// SIMATIC S7-200 project (STEP 7-Micro/WIN), CPU 224 REL 02.01

SYMBOL_TABLE Command
hhhmi_to_plc     VW401
aaa_to_plc       VW402
dor_baraye_1_doff VW320
second_PLC       VW318
minute_PLC       VW316
hour_PLC         VW314
RPM_mani_Cylinder_HMI VW312    // analog_output
RPM_Doffer_Int   VW310    // rpm
RPM_main_Int     VW308    // rpm
RPM_Feed_in_HMI  VW306    // analog_output
RPM_Coiler_In_HMI VW304    // analog_output
RPM_Sec_Cyli_in_HMI VW302    // analog_output
RPM_Doffer_in_HMI VW300    // analog_output
Minute_shiftC    VW248    // amar
hour_shiftC      VW246    // amar
minute_shiftB    VW244    // amar
Lengh            VW242    // doff
max_rpm_SecCylindr VW240    // analog_output
max_rpm_feeder   VW238    // analog_output
max_rpm_coiler   VW236    // analog_output
max_rpm_doffer_cylinder VW234    // analog_output
max_rpm_main_cylinder VW232    // rpm
zaribe_asli_doffer VW230    // rpm
hour_shiftB      VW228    // amar
doff_in_shiftc   VW224    // amar
Minute_ShiftA    VW222    // amar
doff_in_shiftB   VW218    // amar
hour_ShiftA      VW216    // amar
doff_in_shiftA   VW212    // amar
enter_rpm_in_HMI VW210    // analog_output
Zaribe_Asli      VW208    // rpm
Zaribe_Fed       VW206    // analog_output
Zaribe_Coi       VW204    // analog_output
Zaribe_Sec       VW202    // analog_output
Zaribe_Doff      VW200    // analog_output
zaribe_asli2     VD800
leng_for_1rotate_coiler VD720    // doff
Vazne_kole_C     VD712
Vazne_kole_B     VD708
vazne_kole_A     VD704
nomre_fetile     VD700
RPM_Main         VD504
RPM_Doffer       VD500
reset_metal      V104.1
metal_blink_hmi  V104.0
metal_hmi        V103.7
fault            V103.6
coiler_fault     V103.5   // startstop
Metal            V103.4   // startstop
Pulse            V103.3   // pulse_700ms
Doff_Lamp_F      V103.2   // doff
reset_lengh      V103.1   // doff
reset_Amar       V103.0
photocell_coiler_fault V101.6
key_stop_pushed  V101.1   // alarm
Machin_Fault     V101.0   // alarm
OL_Za_F          V100.7   // alarm
OL_ap_F          V100.6   // alarm
OL_Chane_F       V100.5   // alarm
Fauklt_CoilerDrive_F V100.4   // alarm
Fault_FeederDrive_F V100.3   // alarm
Fault_DofferDrive_F V100.2   // alarm
Fault_secDrive_F V100.1   // alarm
fault_mainDrive_F V100.0   // alarm
delay_300ms      T63
metal            T62
timer_for_metal  T61
time_for_push_stop T60
timer_for_coilerfult T59      // start_stop
timer_for_metaldetector T58      // start_stop
Timer57          T57
Timer56          T56
delay            T55      // doff
timer_for_reset_lengh T54      // doff
Timer_for_fan2   T53      // fan
timer_for_fan1   T52      // fan
Stop_Apron       T51      // hopper
for_start_apron  T50      // hopper
Ajir_metal       Q2.5
Fan2             Q2.4
Orange_Lamp      Q2.2
Red_Lamp         Q2.1
Green_Lamp       Q2.0
Feeder_Reverse   Q1.1
Fan1             Q1.0
Zanandeh         Q0.7
Apron            Q0.6
motor_Change_Doff Q0.5
motor_Feeder_Forward Q0.4
motor_Coiler     Q0.3
motor_Doffer     Q0.2
Secondary        Q0.1
Main_Sylinder    Q0.0
Chaper_fault     I2.5
manual_doff      I2.4
OL_Zanandeh      I2.3
OL_Apron         I2.2
OL_change_doff   I2.1
Photocell        I2.0
photocell_coiler I1.5
Fault_Feeder_Drive I1.4
Fault_Coiler_Drive I1.3
Fault_Doffer_Drive I1.2
Fault_Secondary_Drive I1.1
Fault_MainDrive  I1.0
MetalDetector    I0.7
Motor_Doff_SW    I0.5
Emergency        I0.4
Stopp            I0.3
Start            I0.2
Product_SW       I0.1
Hour_counter     C4       // amar
Minute_Counter   C3       // amar
Scond_counter    C2
doff_counter     C1       // amar
lengh_counter    C0
An_Feeder        AQW8
An_Doffer        AQW6
An_Coiler        AQW4
An_Seco_Syl      AQW2
An_Main_Syl      AQW0
                 ?0_40_0  // pulse_700ms
                 ?0_40_0  // pulse_700ms
                 ?0_40_0  // amar
                 ?0_40_0  // amar
                 ?0_40_0  // amar
END_SYMBOL_TABLE

ORGANIZATION_BLOCK Main:OB1
TITLE=vw200 & vw300  -------   vd700 & vd900 ======>> retentive
// vw300 & vw & vw500   ,   vd500 & vd700 =====>not retentive
// vw100 & vw200  ====>> flag
BEGIN
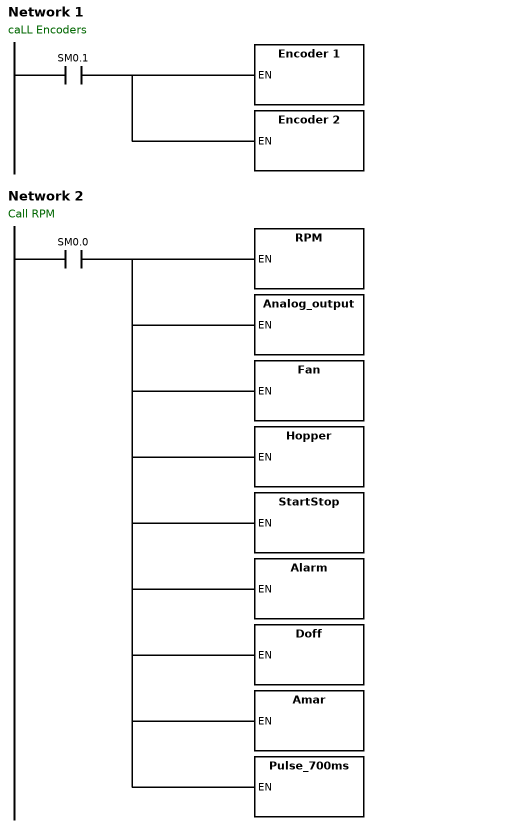
Network 1
// caLL Encoders
LD     SM0.1
CALL   Encoder 1:SBR1
CALL   Encoder 2:SBR2
Network 2
// Call RPM
LD     SM0.0
CALL   RPM:SBR3
CALL   Analog_output:SBR4
CALL   Fan:SBR5
CALL   Hopper:SBR6
CALL   StartStop:SBR8
CALL   Alarm:SBR7
CALL   Doff:SBR9
CALL   Amar:SBR10
CALL   Pulse_700ms:SBR11
END_ORGANIZATION_BLOCK

SUBROUTINE_BLOCK PtoRPM:SBR0
TITLE=子程序注释
VAR_INPUT
Plus:DWORD;	// LD0 
Lines:DWORD;	// LD4 
END_VAR
VAR_IN_OUT
Plusbefore:DWORD;	// LD8 
END_VAR
VAR_OUTPUT
RpmofEncoder:DWORD;	// LD12 
END_VAR
BEGIN
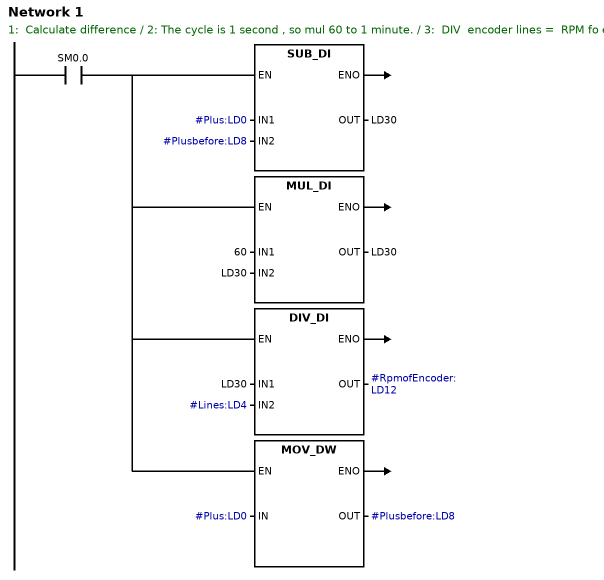
Network 1
// 1:  Calculate difference
// 2: The cycle is 1 second , so mul 60 to 1 minute.
// 3:  DIV  encoder lines =  RPM fo encoder
// 4: save plus to plusbefore
LD     SM0.0
MOVD   #Plus:LD0, LD30
-D     #Plusbefore:LD8, LD30
*D     60, LD30
MOVD   LD30, #RpmofEncoder:LD12
/D     #Lines:LD4, #RpmofEncoder:LD12
MOVD   #Plus:LD0, #Plusbefore:LD8
END_SUBROUTINE_BLOCK

SUBROUTINE_BLOCK Encoder 1:SBR1
TITLE=
BEGIN
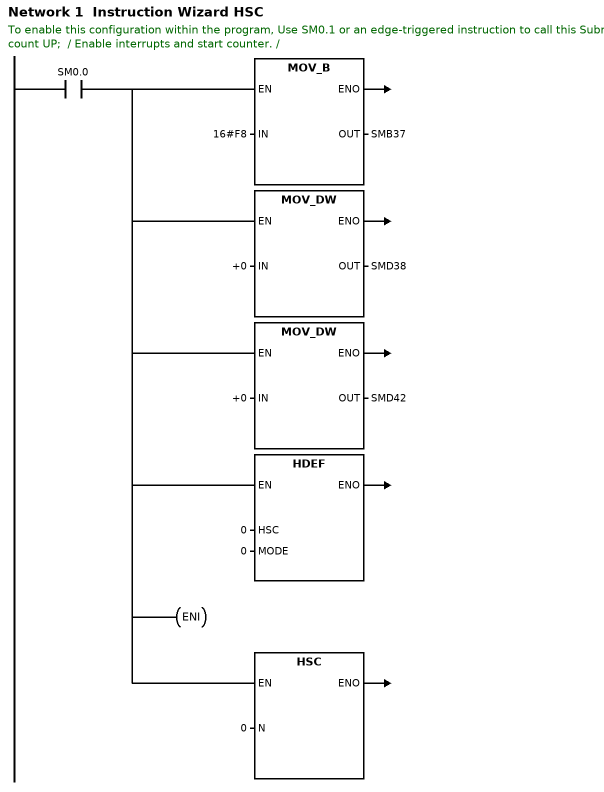
Network 1 // Instruction Wizard HSC
// To enable this configuration within the program, Use SM0.1 or an edge-triggered instruction to call this Subroutine once from the MAIN program block.  
// Configure HC0 for Mode 0; CV = 0; PV = 0; count UP; 
// Enable interrupts and start counter.
// 
//Set control bits: count UP; enabled; 
//Load CV
//Load PV
LD     SM0.0
MOVB   16#F8, SMB37
MOVD   +0, SMD38
MOVD   +0, SMD42
HDEF   0, 0
ENI
HSC    0
END_SUBROUTINE_BLOCK

SUBROUTINE_BLOCK Encoder 2:SBR2
TITLE=
BEGIN
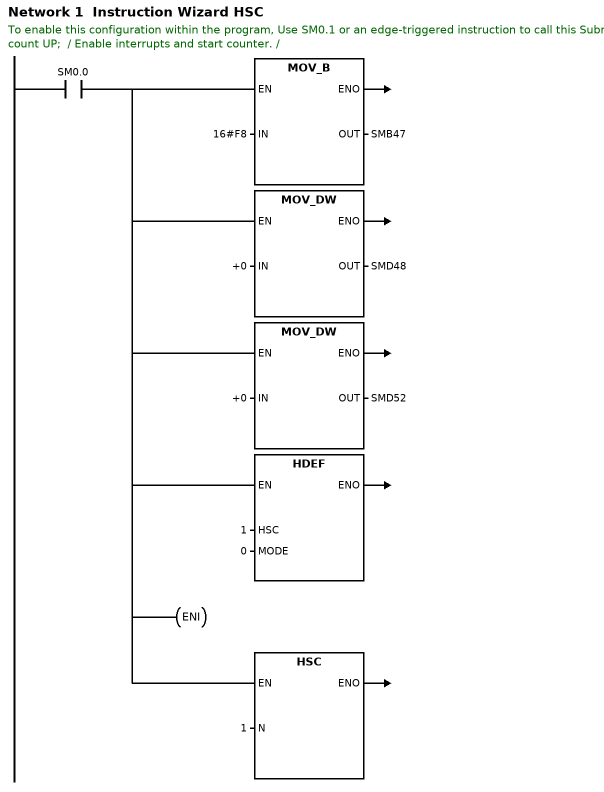
Network 1 // Instruction Wizard HSC
// To enable this configuration within the program, Use SM0.1 or an edge-triggered instruction to call this Subroutine once from the MAIN program block.  
// Configure HC1 for Mode 0; CV = 0; PV = 0; count UP; 
// Enable interrupts and start counter.
// 
//Set control bits: count UP; enabled; 
//Load CV
//Load PV
LD     SM0.0
MOVB   16#F8, SMB47
MOVD   +0, SMD48
MOVD   +0, SMD52
HDEF   1, 0
ENI
HSC    1
END_SUBROUTINE_BLOCK

SUBROUTINE_BLOCK RPM:SBR3
TITLE=SUBROUTINE COMMENTS
VAR
rpm1:REAL;	// LD0 
rpm2:REAL;	// LD4 
rpm11:REAL;	// LD8 
rpm21:REAL;	// LD12 
END_VAR
BEGIN
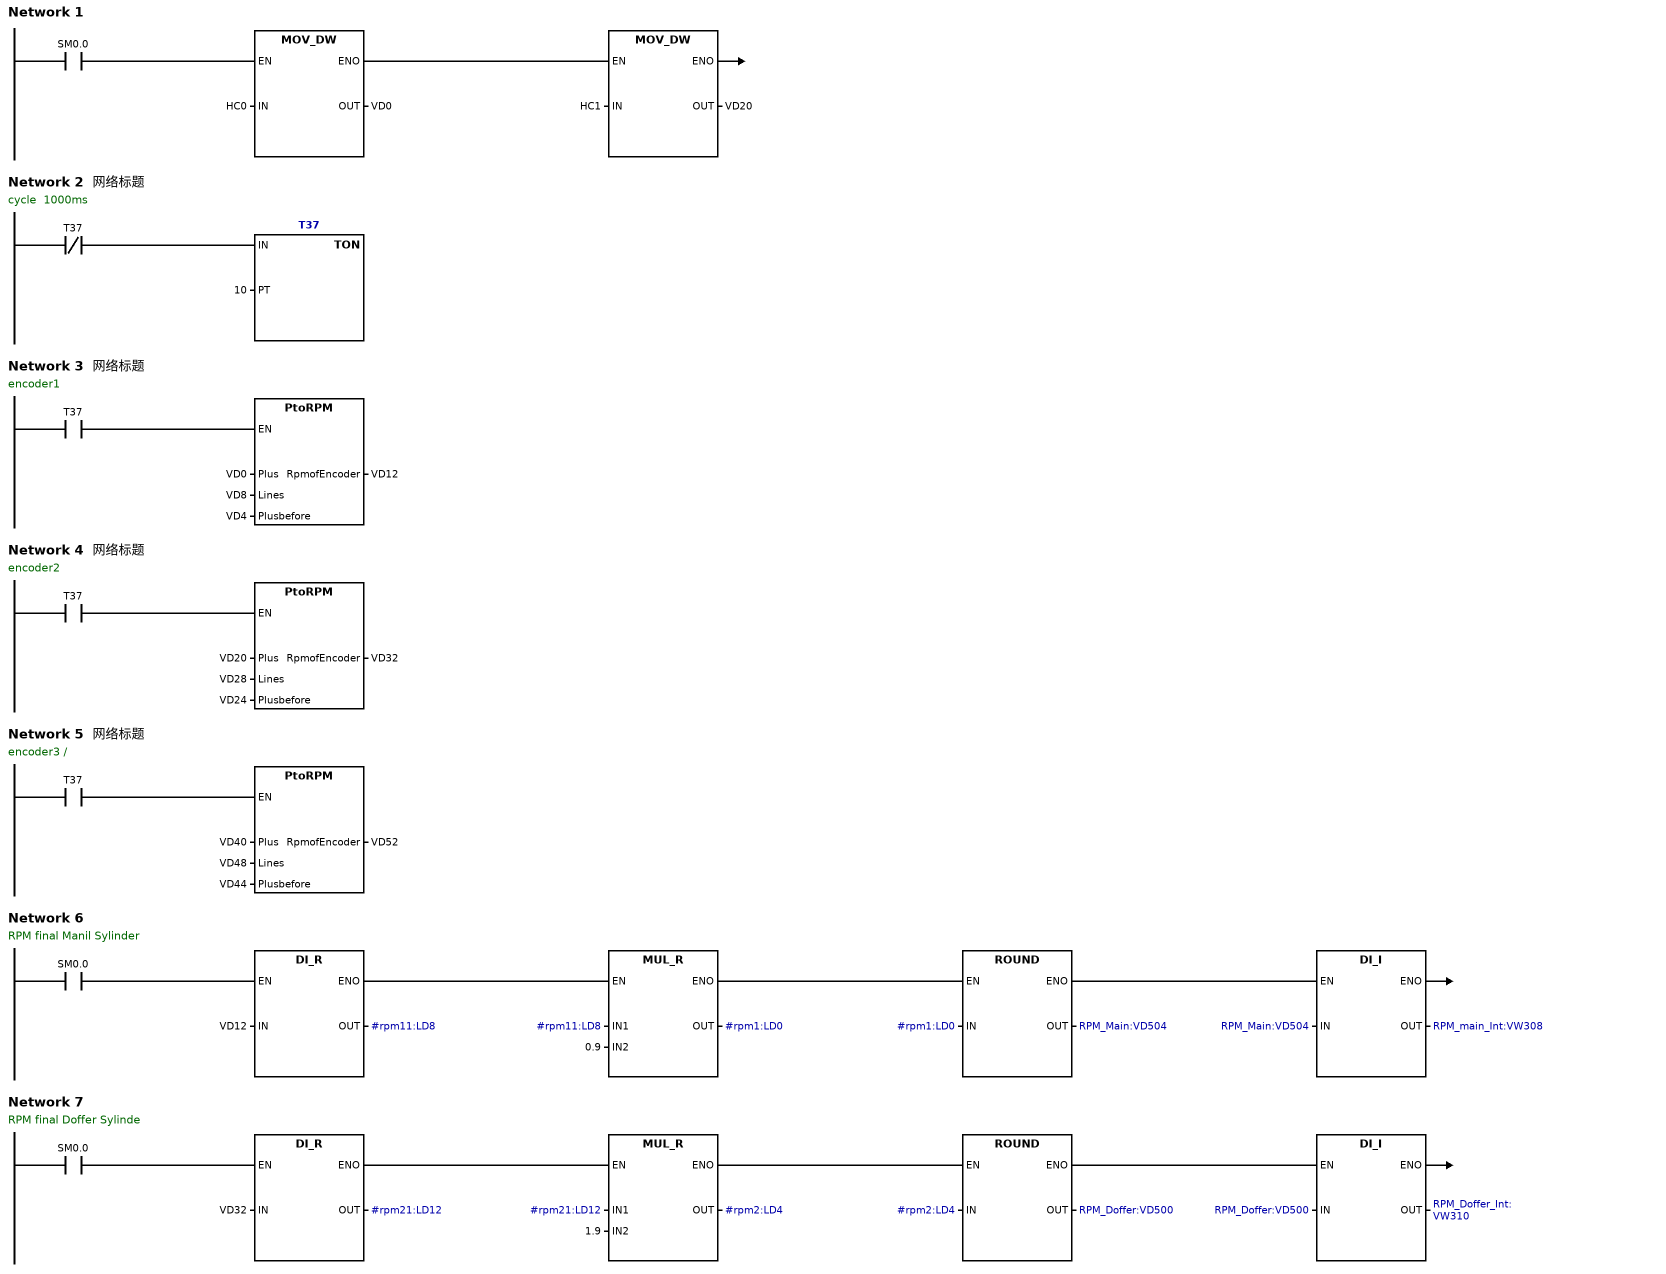
Network 1
LD     SM0.0
MOVD   HC0, VD0
AENO
MOVD   HC1, VD20
Network 2 // 网络标题
// cycle  1000ms 
LDN    T37
TON    T37, 10
Network 3 // 网络标题
// encoder1
LD     T37
CALL   PtoRPM:SBR0, VD0, VD8, VD4, VD12
Network 4 // 网络标题
// encoder2
LD     T37
CALL   PtoRPM:SBR0, VD20, VD28, VD24, VD32
Network 5 // 网络标题
// encoder3
// 
LD     T37
CALL   PtoRPM:SBR0, VD40, VD48, VD44, VD52
Network 6
// RPM final Manil Sylinder
LD     SM0.0
DTR    VD12, #rpm11:LD8
AENO
MOVR   #rpm11:LD8, #rpm1:LD0
AENO
*R     0.9, #rpm1:LD0
AENO
ROUND  #rpm1:LD0, RPM_Main:VD504
AENO
DTI    RPM_Main:VD504, RPM_main_Int:VW308
Network 7
// RPM final Doffer Sylinde
LD     SM0.0
DTR    VD32, #rpm21:LD12
AENO
MOVR   #rpm21:LD12, #rpm2:LD4
AENO
*R     1.9, #rpm2:LD4
AENO
ROUND  #rpm2:LD4, RPM_Doffer:VD500
AENO
DTI    RPM_Doffer:VD500, RPM_Doffer_Int:VW310
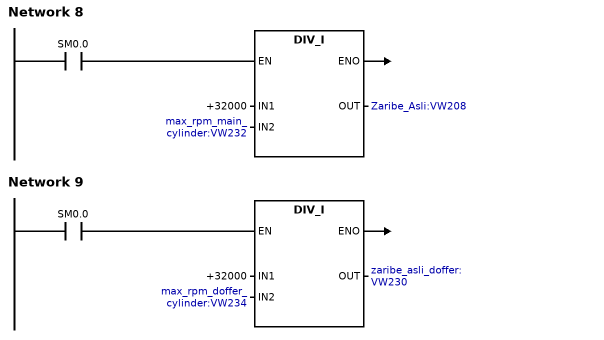
Network 8
LD     SM0.0
MOVW   +32000, Zaribe_Asli:VW208
/I     max_rpm_main_cylinder:VW232, Zaribe_Asli:VW208
Network 9
LD     SM0.0
MOVW   +32000, zaribe_asli_doffer:VW230
/I     max_rpm_doffer_cylinder:VW234, zaribe_asli_doffer:VW230
END_SUBROUTINE_BLOCK

SUBROUTINE_BLOCK Analog_output:SBR4
TITLE=SUBROUTINE COMMENTS
VAR
rpm_doff1:DINT;	// LD0 
rpm_doff2:DINT;	// LD4 
rpm_doff3:INT;	// LW8 
rpm_sec1:INT;	// LW10 
rpm_sec2:INT;	// LW12 
rpm_sec3:INT;	// LW14 
rpm_coil1:INT;	// LW16 
rpm_coil2:INT;	// LW18 
rpm_coil3:INT;	// LW20 
ADD:INT;	// LW22 
rpm_feed2:INT;	// LW24 
rpm_feed3:INT;	// LW26 
speed_main:INT;	// LW28 
main_hmi1:INT;	// LW30 
main_hmi2:INT;	// LW32 
dofer_hmi1:INT;	// LW34 
dofer_hmi2:INT;	// LW36 
sec_hmi1:INT;	// LW38 
sec_hmi2:INT;	// LW40 
coiler_hmi1:INT;	// LW42 
coiler_hmi2:INT;	// LW44 
feeder_hmi1:INT;	// LW46 
feeder_hmi2:INT;	// LW48 
rmp_doffer1:DINT;	// LD50 
rpm_doffer2:DINT;	// LD54 
END_VAR
BEGIN
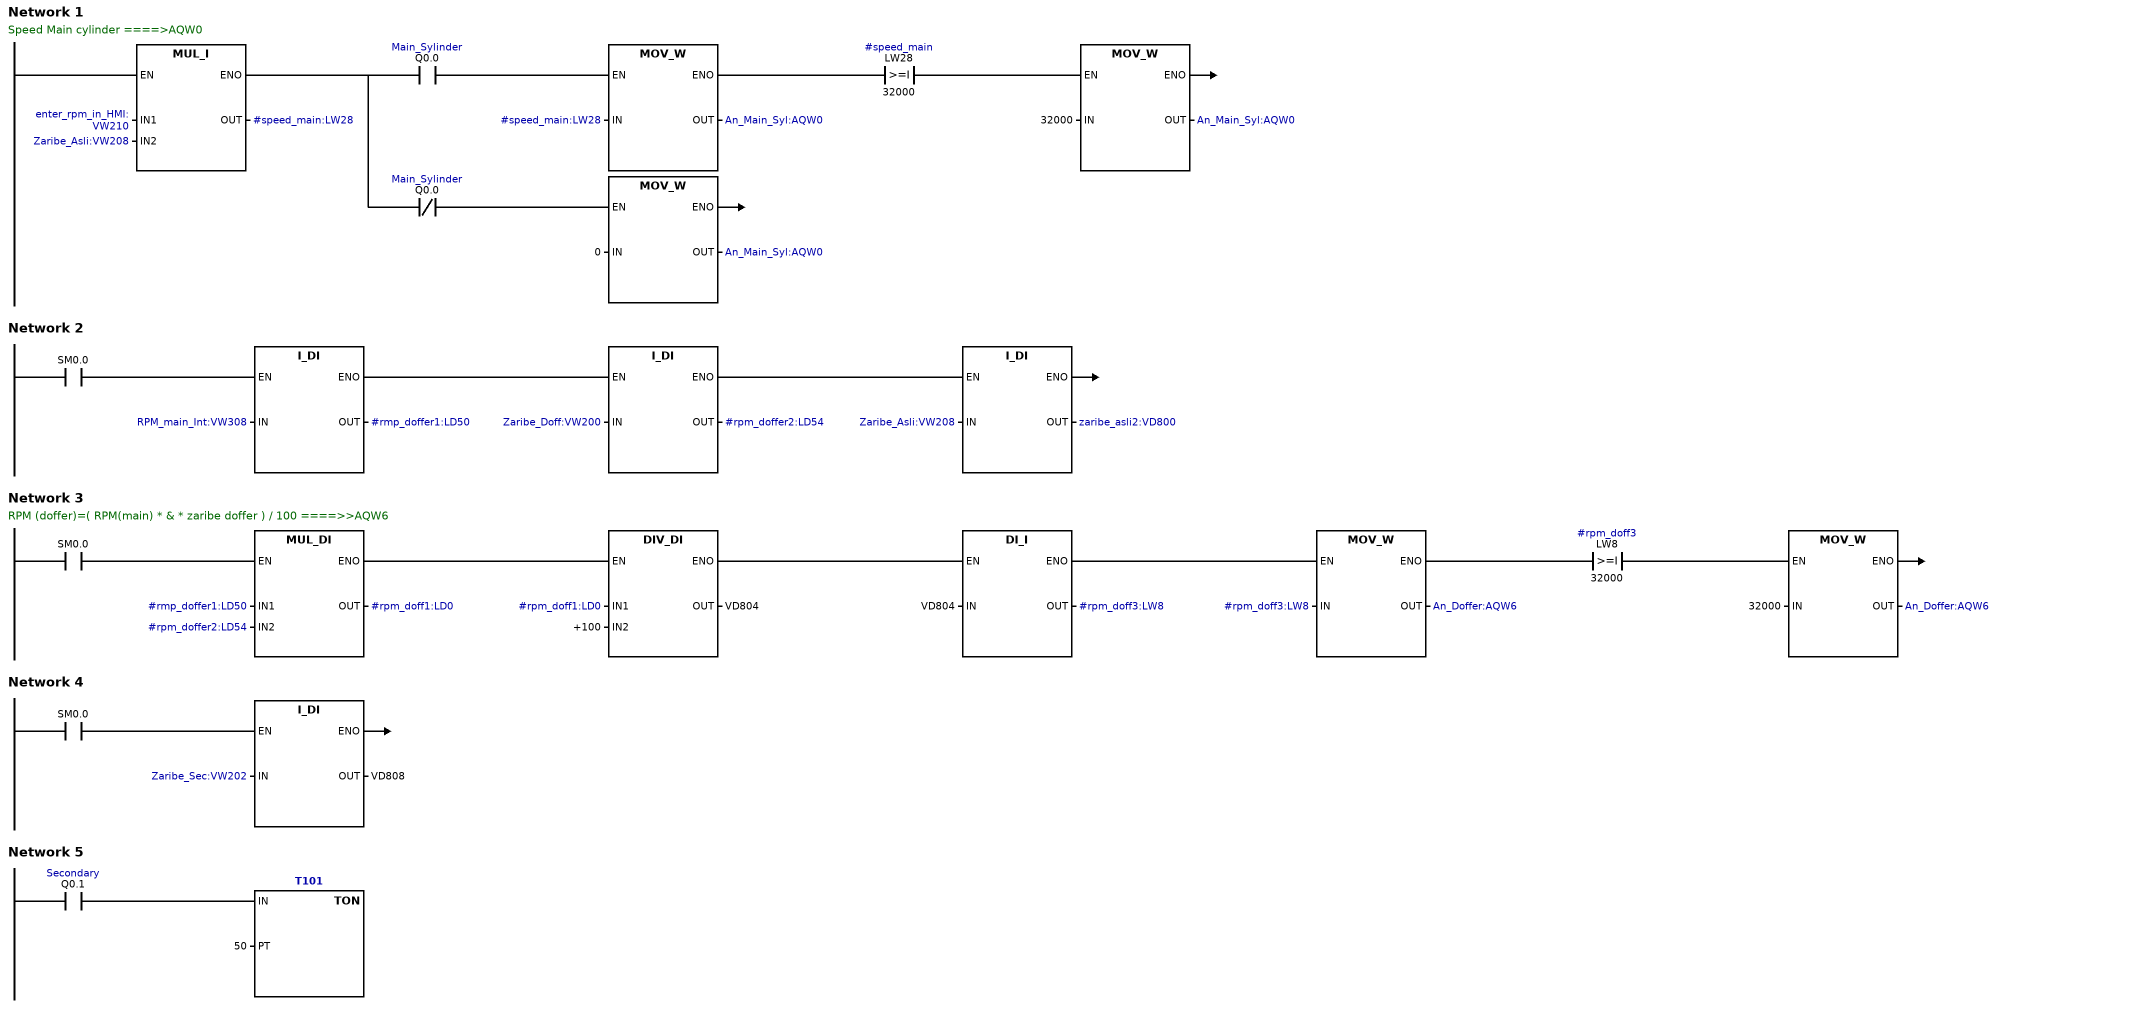
Network 1
// Speed Main cylinder ====>AQW0
MOVW   enter_rpm_in_HMI:VW210, #speed_main:LW28
AENO
*I     Zaribe_Asli:VW208, #speed_main:LW28
AENO
LPS
A      Main_Sylinder:Q0.0
MOVW   #speed_main:LW28, An_Main_Syl:AQW0
AENO
AW>=   #speed_main:LW28, 32000
MOVW   32000, An_Main_Syl:AQW0
LPP
AN     Main_Sylinder:Q0.0
MOVW   0, An_Main_Syl:AQW0
Network 2
LD     SM0.0
ITD    RPM_main_Int:VW308, #rmp_doffer1:LD50
AENO
ITD    Zaribe_Doff:VW200, #rpm_doffer2:LD54
AENO
ITD    Zaribe_Asli:VW208, zaribe_asli2:VD800
Network 3
// RPM (doffer)=( RPM(main) * & * zaribe doffer ) / 100 ====>>AQW6
LD     SM0.0
MOVD   #rmp_doffer1:LD50, #rpm_doff1:LD0
AENO
*D     #rpm_doffer2:LD54, #rpm_doff1:LD0
AENO
MOVD   #rpm_doff1:LD0, VD804
AENO
/D     +100, VD804
AENO
DTI    VD804, #rpm_doff3:LW8
AENO
MOVW   #rpm_doff3:LW8, An_Doffer:AQW6
AENO
AW>=   #rpm_doff3:LW8, 32000
MOVW   32000, An_Doffer:AQW6
Network 4
LD     SM0.0
ITD    Zaribe_Sec:VW202, VD808
Network 5
LD     Secondary:Q0.1
TON    T101, 50
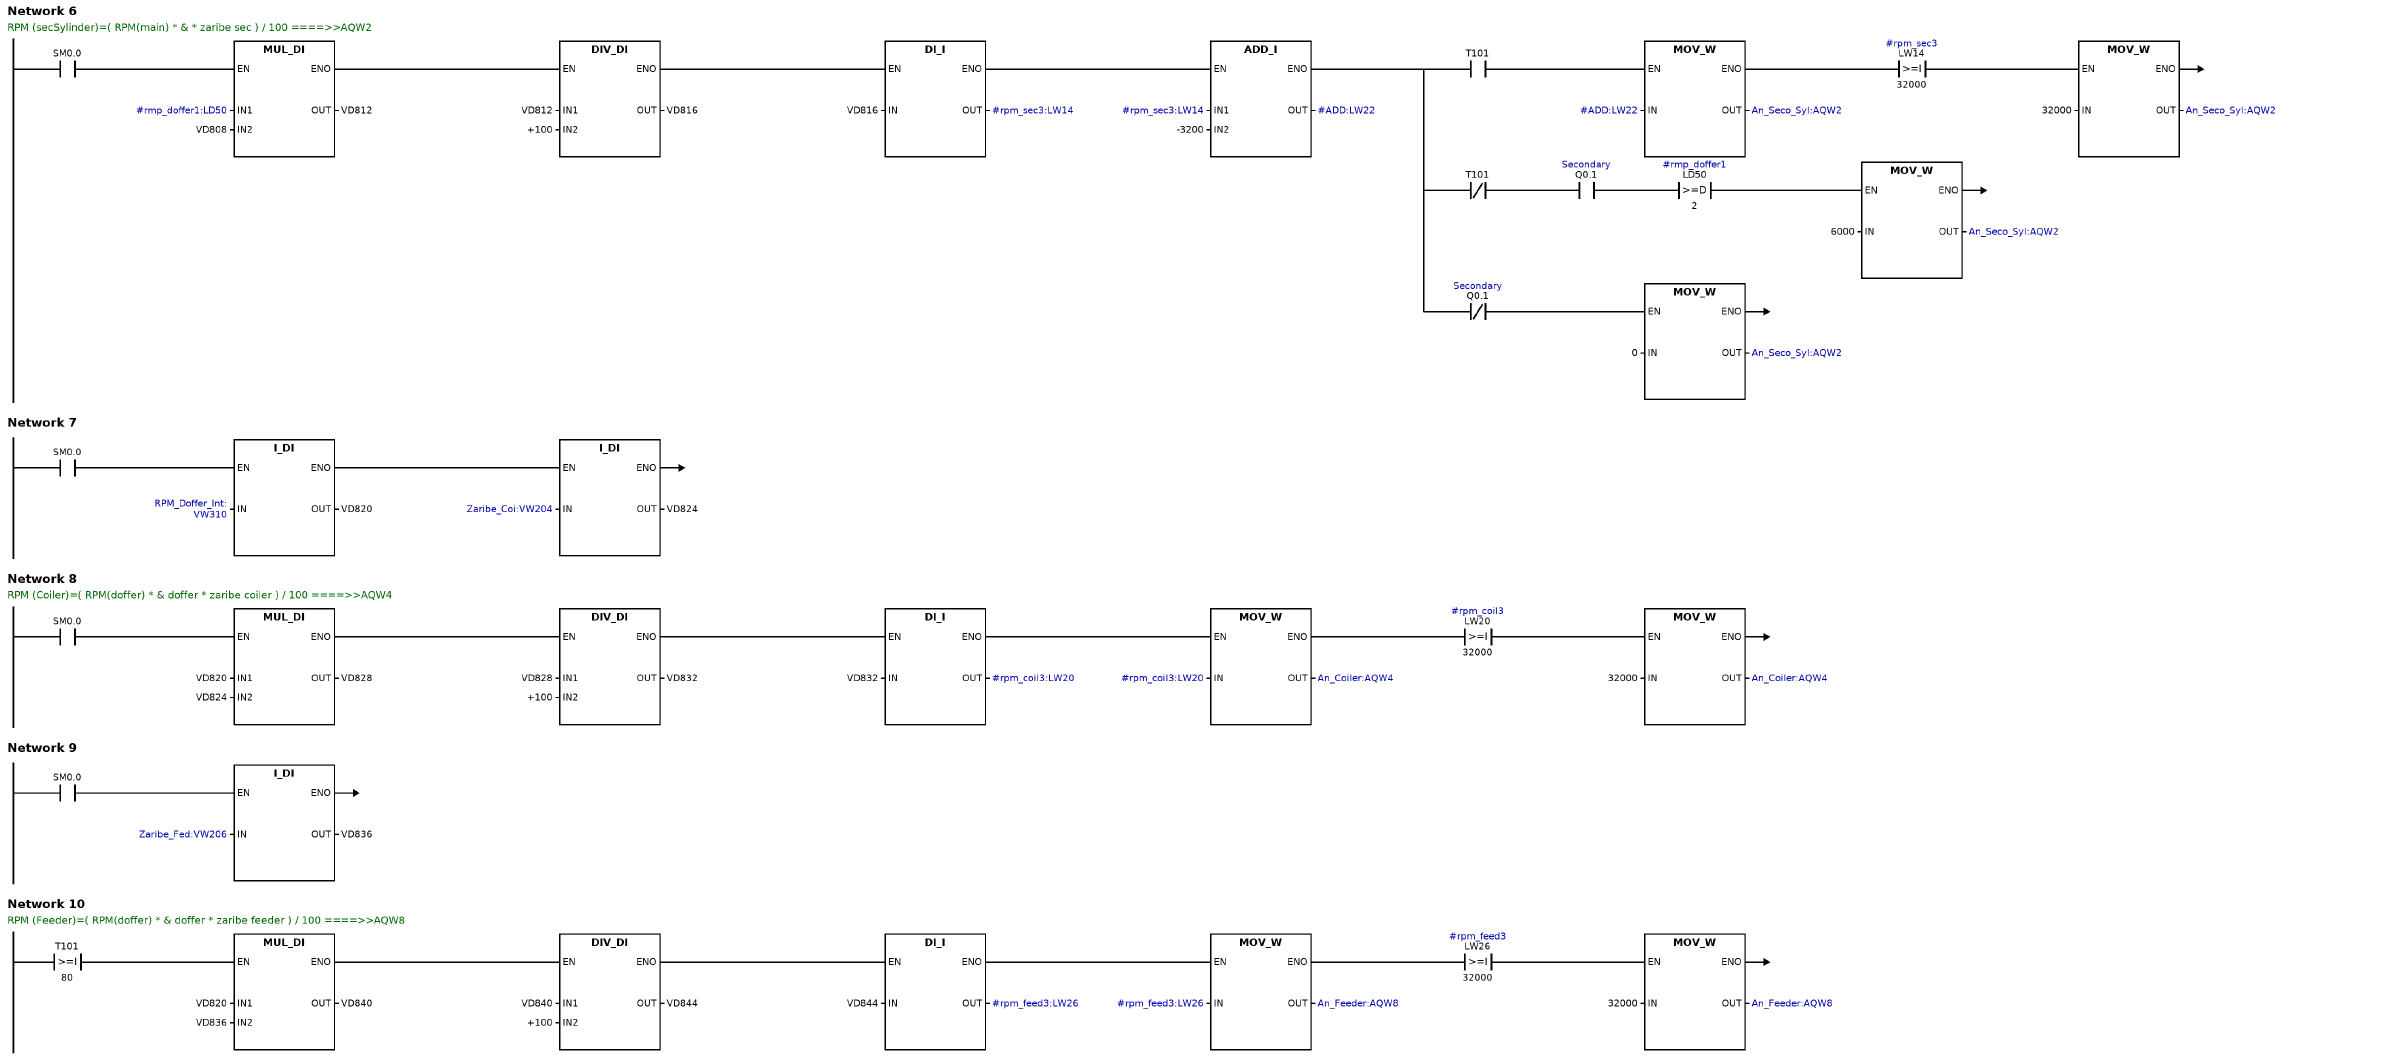
Network 6
// RPM (secSylinder)=( RPM(main) * & * zaribe sec ) / 100 ====>>AQW2
LD     SM0.0
MOVD   #rmp_doffer1:LD50, VD812
AENO
*D     VD808, VD812
AENO
MOVD   VD812, VD816
AENO
/D     +100, VD816
AENO
DTI    VD816, #rpm_sec3:LW14
AENO
MOVW   #rpm_sec3:LW14, #ADD:LW22
AENO
+I     -3200, #ADD:LW22
AENO
LPS
A      T101
MOVW   #ADD:LW22, An_Seco_Syl:AQW2
AENO
AW>=   #rpm_sec3:LW14, 32000
MOVW   32000, An_Seco_Syl:AQW2
LRD
AN     T101
A      Secondary:Q0.1
AD>=   #rmp_doffer1:LD50, 2
MOVW   6000, An_Seco_Syl:AQW2
LPP
AN     Secondary:Q0.1
MOVW   0, An_Seco_Syl:AQW2
Network 7
LD     SM0.0
ITD    RPM_Doffer_Int:VW310, VD820
AENO
ITD    Zaribe_Coi:VW204, VD824
Network 8
// RPM (Coiler)=( RPM(doffer) * & doffer * zaribe coiler ) / 100 ====>>AQW4
LD     SM0.0
MOVD   VD820, VD828
AENO
*D     VD824, VD828
AENO
MOVD   VD828, VD832
AENO
/D     +100, VD832
AENO
DTI    VD832, #rpm_coil3:LW20
AENO
MOVW   #rpm_coil3:LW20, An_Coiler:AQW4
AENO
AW>=   #rpm_coil3:LW20, 32000
MOVW   32000, An_Coiler:AQW4
Network 9
LD     SM0.0
ITD    Zaribe_Fed:VW206, VD836
Network 10
// RPM (Feeder)=( RPM(doffer) * & doffer * zaribe feeder ) / 100 ====>>AQW8
LDW>=  T101, 80
MOVD   VD820, VD840
AENO
*D     VD836, VD840
AENO
MOVD   VD840, VD844
AENO
/D     +100, VD844
AENO
DTI    VD844, #rpm_feed3:LW26
AENO
MOVW   #rpm_feed3:LW26, An_Feeder:AQW8
AENO
AW>=   #rpm_feed3:LW26, 32000
MOVW   32000, An_Feeder:AQW8
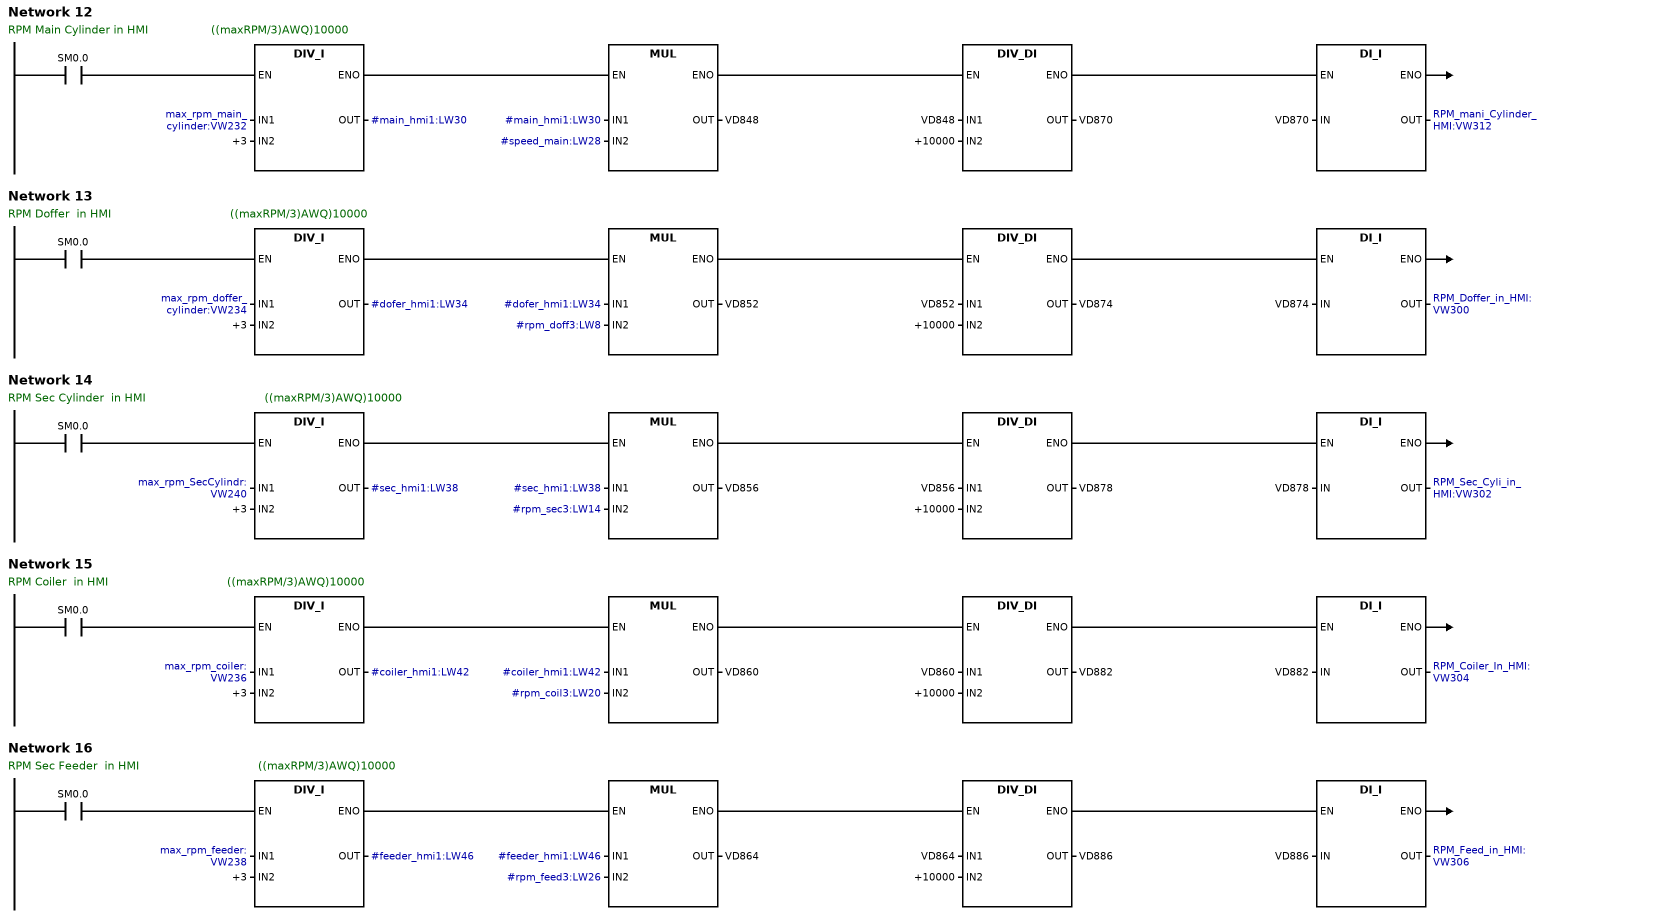
Network 12
// RPM Main Cylinder in HMI                  ((maxRPM/3)AWQ)10000
LD     SM0.0
MOVW   max_rpm_main_cylinder:VW232, #main_hmi1:LW30
AENO
/I     +3, #main_hmi1:LW30
AENO
MOVW   #main_hmi1:LW30, VW850
AENO
MUL    #speed_main:LW28, VD848
AENO
MOVD   VD848, VD870
AENO
/D     +10000, VD870
AENO
DTI    VD870, RPM_mani_Cylinder_HMI:VW312
Network 13
// RPM Doffer  in HMI                                  ((maxRPM/3)AWQ)10000
LD     SM0.0
MOVW   max_rpm_doffer_cylinder:VW234, #dofer_hmi1:LW34
AENO
/I     +3, #dofer_hmi1:LW34
AENO
MOVW   #dofer_hmi1:LW34, VW854
AENO
MUL    #rpm_doff3:LW8, VD852
AENO
MOVD   VD852, VD874
AENO
/D     +10000, VD874
AENO
DTI    VD874, RPM_Doffer_in_HMI:VW300
Network 14
// RPM Sec Cylinder  in HMI                                  ((maxRPM/3)AWQ)10000
LD     SM0.0
MOVW   max_rpm_SecCylindr:VW240, #sec_hmi1:LW38
AENO
/I     +3, #sec_hmi1:LW38
AENO
MOVW   #sec_hmi1:LW38, VW858
AENO
MUL    #rpm_sec3:LW14, VD856
AENO
MOVD   VD856, VD878
AENO
/D     +10000, VD878
AENO
DTI    VD878, RPM_Sec_Cyli_in_HMI:VW302
Network 15
// RPM Coiler  in HMI                                  ((maxRPM/3)AWQ)10000
LD     SM0.0
MOVW   max_rpm_coiler:VW236, #coiler_hmi1:LW42
AENO
/I     +3, #coiler_hmi1:LW42
AENO
MOVW   #coiler_hmi1:LW42, VW862
AENO
MUL    #rpm_coil3:LW20, VD860
AENO
MOVD   VD860, VD882
AENO
/D     +10000, VD882
AENO
DTI    VD882, RPM_Coiler_In_HMI:VW304
Network 16
// RPM Sec Feeder  in HMI                                  ((maxRPM/3)AWQ)10000
LD     SM0.0
MOVW   max_rpm_feeder:VW238, #feeder_hmi1:LW46
AENO
/I     +3, #feeder_hmi1:LW46
AENO
MOVW   #feeder_hmi1:LW46, VW866
AENO
MUL    #rpm_feed3:LW26, VD864
AENO
MOVD   VD864, VD886
AENO
/D     +10000, VD886
AENO
DTI    VD886, RPM_Feed_in_HMI:VW306
END_SUBROUTINE_BLOCK

SUBROUTINE_BLOCK Fan:SBR5
TITLE=SUBROUTINE COMMENTS
BEGIN
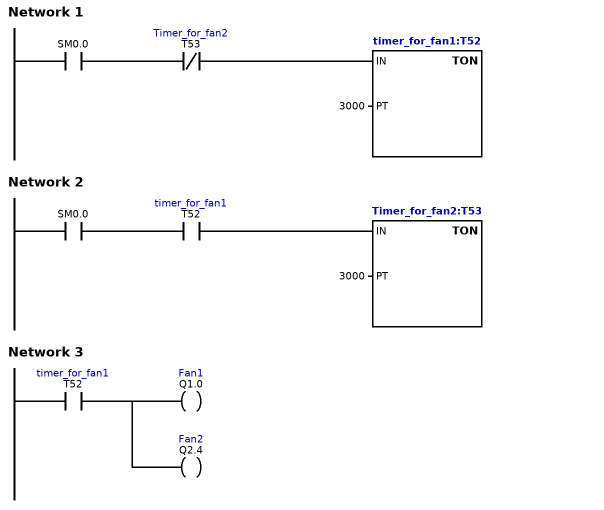
Network 1
LD     SM0.0
AN     Timer_for_fan2:T53
TON    timer_for_fan1:T52, 3000
Network 2
LD     SM0.0
A      timer_for_fan1:T52
TON    Timer_for_fan2:T53, 3000
Network 3
LD     timer_for_fan1:T52
=      Fan1:Q1.0
=      Fan2:Q2.4
Network 4 // Network Title
// Network Comment
END_SUBROUTINE_BLOCK

SUBROUTINE_BLOCK Hopper:SBR6
TITLE=SUBROUTINE COMMENTS
BEGIN
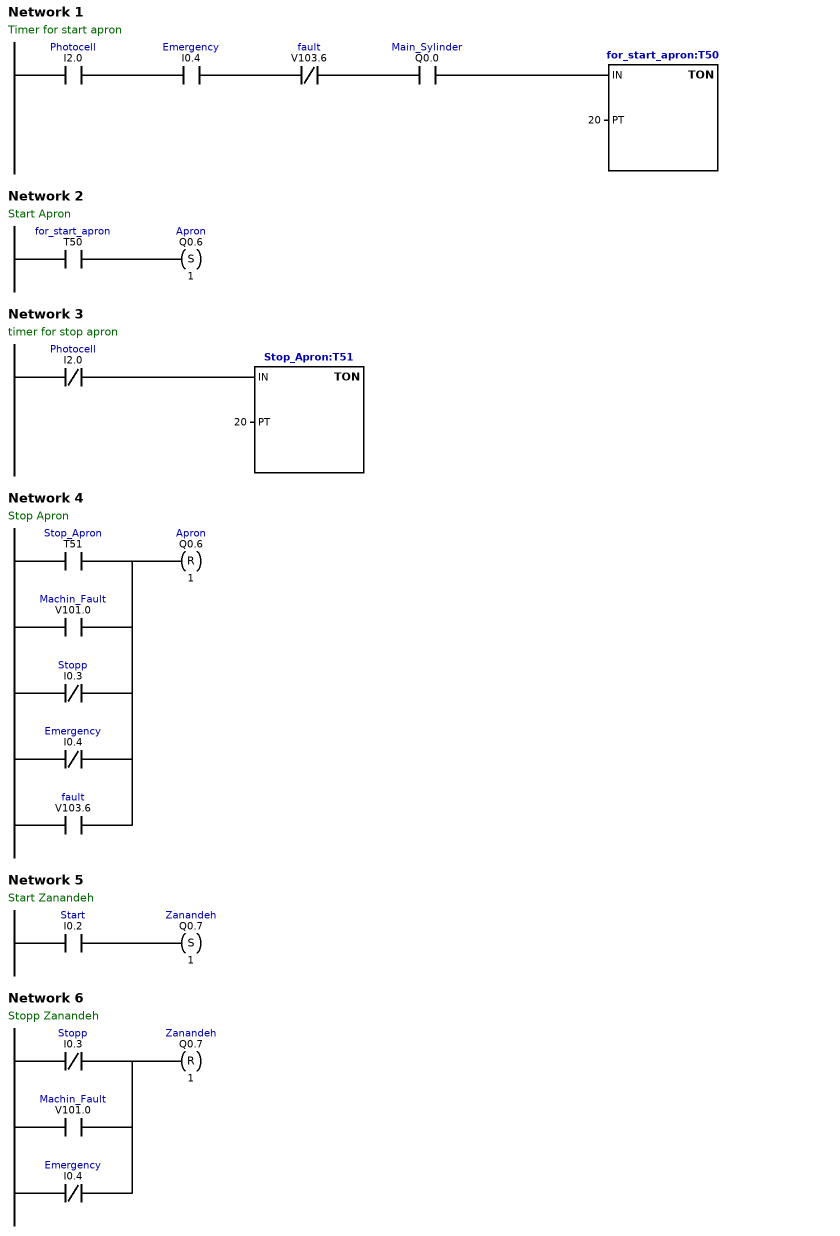
Network 1
// Timer for start apron
LD     Photocell:I2.0
A      Emergency:I0.4
AN     fault:V103.6
A      Main_Sylinder:Q0.0
TON    for_start_apron:T50, 20
Network 2
// Start Apron
LD     for_start_apron:T50
S      Apron:Q0.6, 1
Network 3
// timer for stop apron
LDN    Photocell:I2.0
TON    Stop_Apron:T51, 20
Network 4
// Stop Apron
LD     Stop_Apron:T51
O      Machin_Fault:V101.0
ON     Stopp:I0.3
ON     Emergency:I0.4
O      fault:V103.6
R      Apron:Q0.6, 1
Network 5
// Start Zanandeh
LD     Start:I0.2
S      Zanandeh:Q0.7, 1
Network 6
// Stopp Zanandeh
LDN    Stopp:I0.3
O      Machin_Fault:V101.0
ON     Emergency:I0.4
R      Zanandeh:Q0.7, 1
Network 7 // Network Title
// Network Comment
END_SUBROUTINE_BLOCK

SUBROUTINE_BLOCK Alarm:SBR7
TITLE=SUBROUTINE COMMENTS
BEGIN
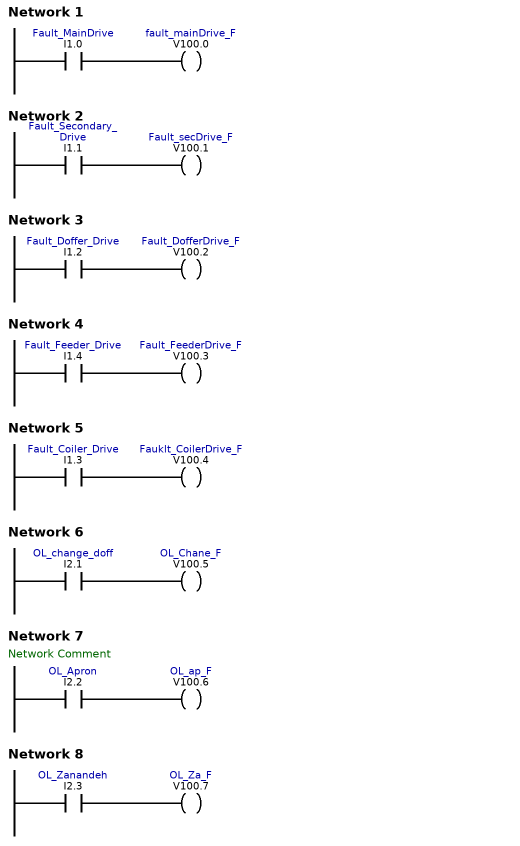
Network 1
LD     Fault_MainDrive:I1.0
=      fault_mainDrive_F:V100.0
Network 2
LD     Fault_Secondary_Drive:I1.1
=      Fault_secDrive_F:V100.1
Network 3
LD     Fault_Doffer_Drive:I1.2
=      Fault_DofferDrive_F:V100.2
Network 4
LD     Fault_Feeder_Drive:I1.4
=      Fault_FeederDrive_F:V100.3
Network 5
LD     Fault_Coiler_Drive:I1.3
=      Fauklt_CoilerDrive_F:V100.4
Network 6
LD     OL_change_doff:I2.1
=      OL_Chane_F:V100.5
Network 7
// Network Comment
LD     OL_Apron:I2.2
=      OL_ap_F:V100.6
Network 8
LD     OL_Zanandeh:I2.3
=      OL_Za_F:V100.7
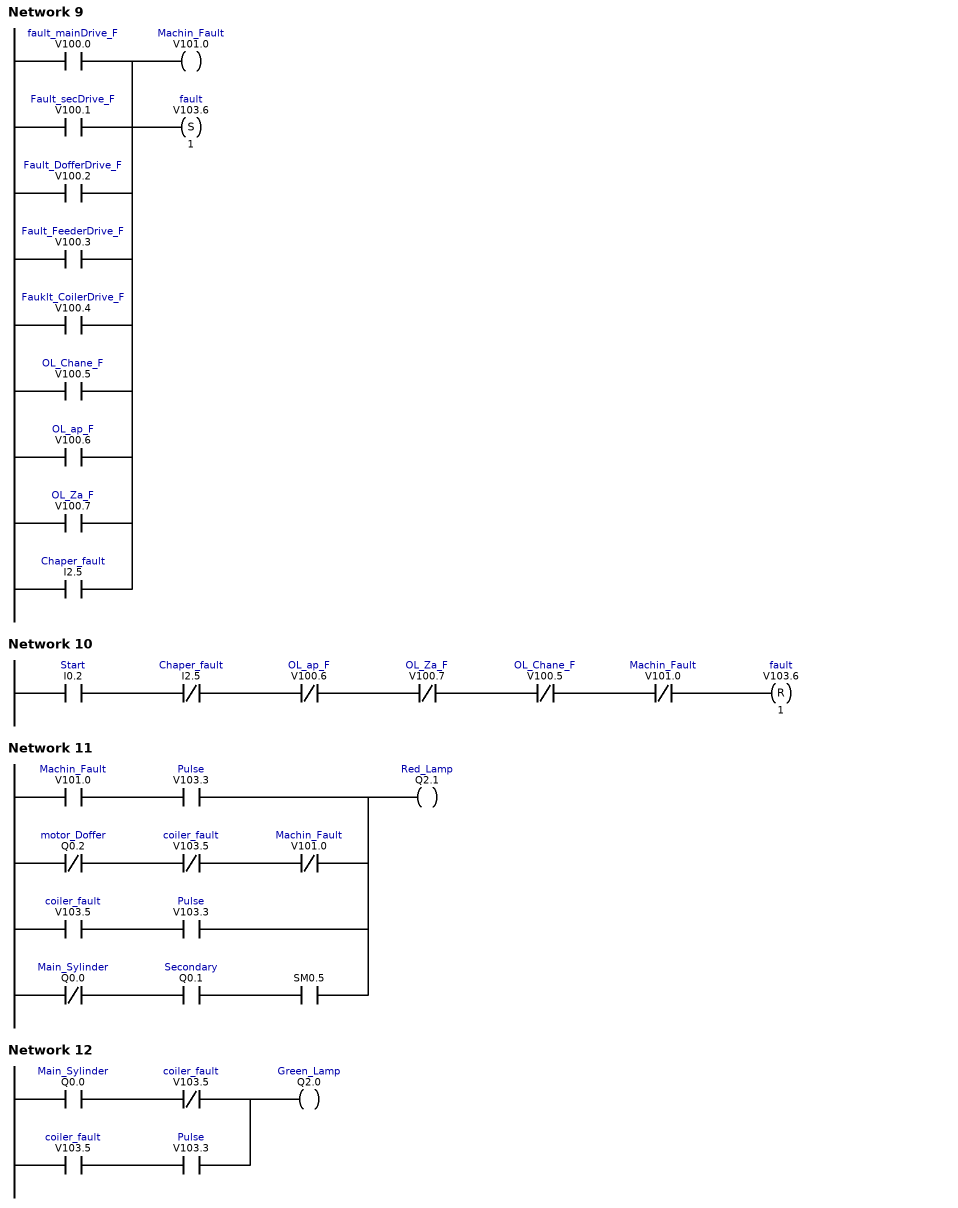
Network 9
LD     fault_mainDrive_F:V100.0
O      Fault_secDrive_F:V100.1
O      Fault_DofferDrive_F:V100.2
O      Fault_FeederDrive_F:V100.3
O      Fauklt_CoilerDrive_F:V100.4
O      OL_Chane_F:V100.5
O      OL_ap_F:V100.6
O      OL_Za_F:V100.7
O      Chaper_fault:I2.5
=      Machin_Fault:V101.0
S      fault:V103.6, 1
Network 10
LD     Start:I0.2
AN     Chaper_fault:I2.5
AN     OL_ap_F:V100.6
AN     OL_Za_F:V100.7
AN     OL_Chane_F:V100.5
AN     Machin_Fault:V101.0
R      fault:V103.6, 1
Network 11
LD     Machin_Fault:V101.0
A      Pulse:V103.3
LDN    motor_Doffer:Q0.2
AN     coiler_fault:V103.5
AN     Machin_Fault:V101.0
OLD
LD     coiler_fault:V103.5
A      Pulse:V103.3
OLD
LDN    Main_Sylinder:Q0.0
A      Secondary:Q0.1
A      SM0.5
OLD
=      Red_Lamp:Q2.1
Network 12
LD     Main_Sylinder:Q0.0
AN     coiler_fault:V103.5
LD     coiler_fault:V103.5
A      Pulse:V103.3
OLD
=      Green_Lamp:Q2.0
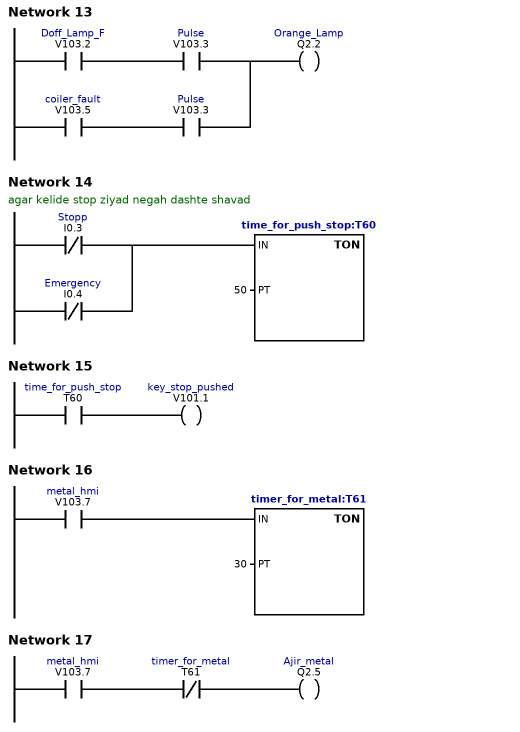
Network 13
LD     Doff_Lamp_F:V103.2
A      Pulse:V103.3
LD     coiler_fault:V103.5
A      Pulse:V103.3
OLD
=      Orange_Lamp:Q2.2
Network 14
// agar kelide stop ziyad negah dashte shavad
LDN    Stopp:I0.3
ON     Emergency:I0.4
TON    time_for_push_stop:T60, 50
Network 15
LD     time_for_push_stop:T60
=      key_stop_pushed:V101.1
Network 16
LD     metal_hmi:V103.7
TON    timer_for_metal:T61, 30
Network 17
LD     metal_hmi:V103.7
AN     timer_for_metal:T61
=      Ajir_metal:Q2.5
END_SUBROUTINE_BLOCK

SUBROUTINE_BLOCK StartStop:SBR8
TITLE=SUBROUTINE COMMENTS
BEGIN
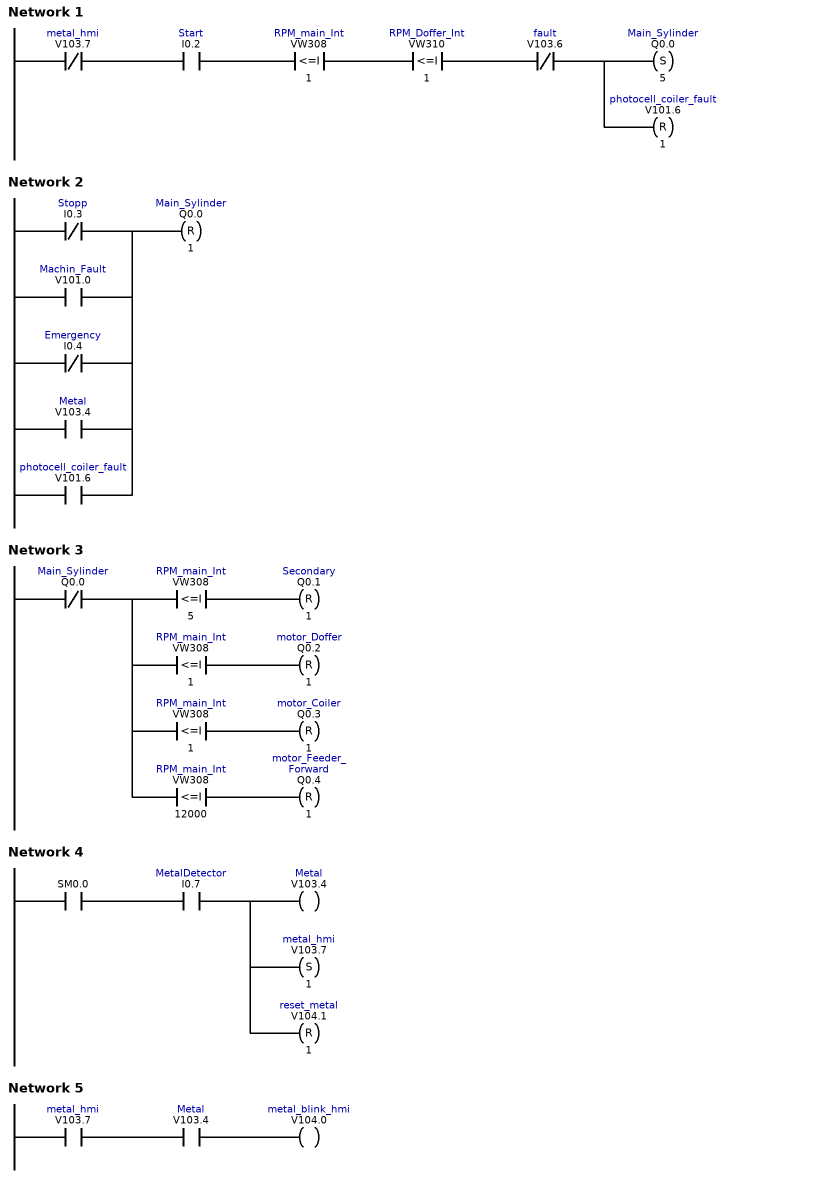
Network 1
LDN    metal_hmi:V103.7
A      Start:I0.2
AW<=   RPM_main_Int:VW308, 1
AW<=   RPM_Doffer_Int:VW310, 1
AN     fault:V103.6
S      Main_Sylinder:Q0.0, 5
R      photocell_coiler_fault:V101.6, 1
Network 2
LDN    Stopp:I0.3
O      Machin_Fault:V101.0
ON     Emergency:I0.4
O      Metal:V103.4
O      photocell_coiler_fault:V101.6
R      Main_Sylinder:Q0.0, 1
Network 3
LDN    Main_Sylinder:Q0.0
LPS
AW<=   RPM_main_Int:VW308, 5
R      Secondary:Q0.1, 1
LRD
AW<=   RPM_main_Int:VW308, 1
R      motor_Doffer:Q0.2, 1
LRD
AW<=   RPM_main_Int:VW308, 1
R      motor_Coiler:Q0.3, 1
LPP
AW<=   RPM_main_Int:VW308, 12000
R      motor_Feeder_Forward:Q0.4, 1
Network 4
LD     SM0.0
A      MetalDetector:I0.7
=      Metal:V103.4
S      metal_hmi:V103.7, 1
R      reset_metal:V104.1, 1
Network 5
// (network saved uncompiled; LAD cells follow)
// row 0: c0 -| |- metal_hmi:V103.7  c1 -| |- Metal:V103.4  c2 -( ) metal_blink_hmi:V104.0
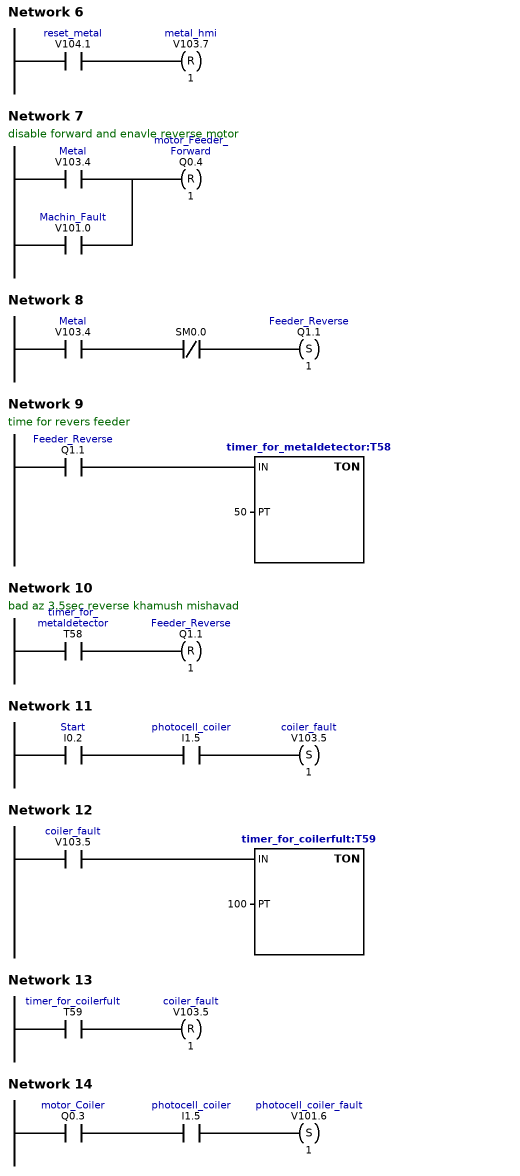
Network 6
LD     reset_metal:V104.1
R      metal_hmi:V103.7, 1
Network 7
// disable forward and enavle reverse motor
LD     Metal:V103.4
O      Machin_Fault:V101.0
R      motor_Feeder_Forward:Q0.4, 1
Network 8
LD     Metal:V103.4
AN     SM0.0
S      Feeder_Reverse:Q1.1, 1
Network 9
// time for revers feeder
LD     Feeder_Reverse:Q1.1
TON    timer_for_metaldetector:T58, 50
Network 10
// bad az 3.5sec reverse khamush mishavad
LD     timer_for_metaldetector:T58
R      Feeder_Reverse:Q1.1, 1
Network 11
LD     Start:I0.2
A      photocell_coiler:I1.5
S      coiler_fault:V103.5, 1
Network 12
LD     coiler_fault:V103.5
TON    timer_for_coilerfult:T59, 100
Network 13
LD     timer_for_coilerfult:T59
R      coiler_fault:V103.5, 1
Network 14
LD     motor_Coiler:Q0.3
A      photocell_coiler:I1.5
S      photocell_coiler_fault:V101.6, 1
END_SUBROUTINE_BLOCK

SUBROUTINE_BLOCK Doff:SBR9
TITLE=SUBROUTINE COMMENTS
VAR
lengh_cm:DINT;	// LD0 
product_DI:DINT;	// LD4 
product_I:INT;	// LW8 
doff1:INT;	// LW10 
END_VAR
BEGIN
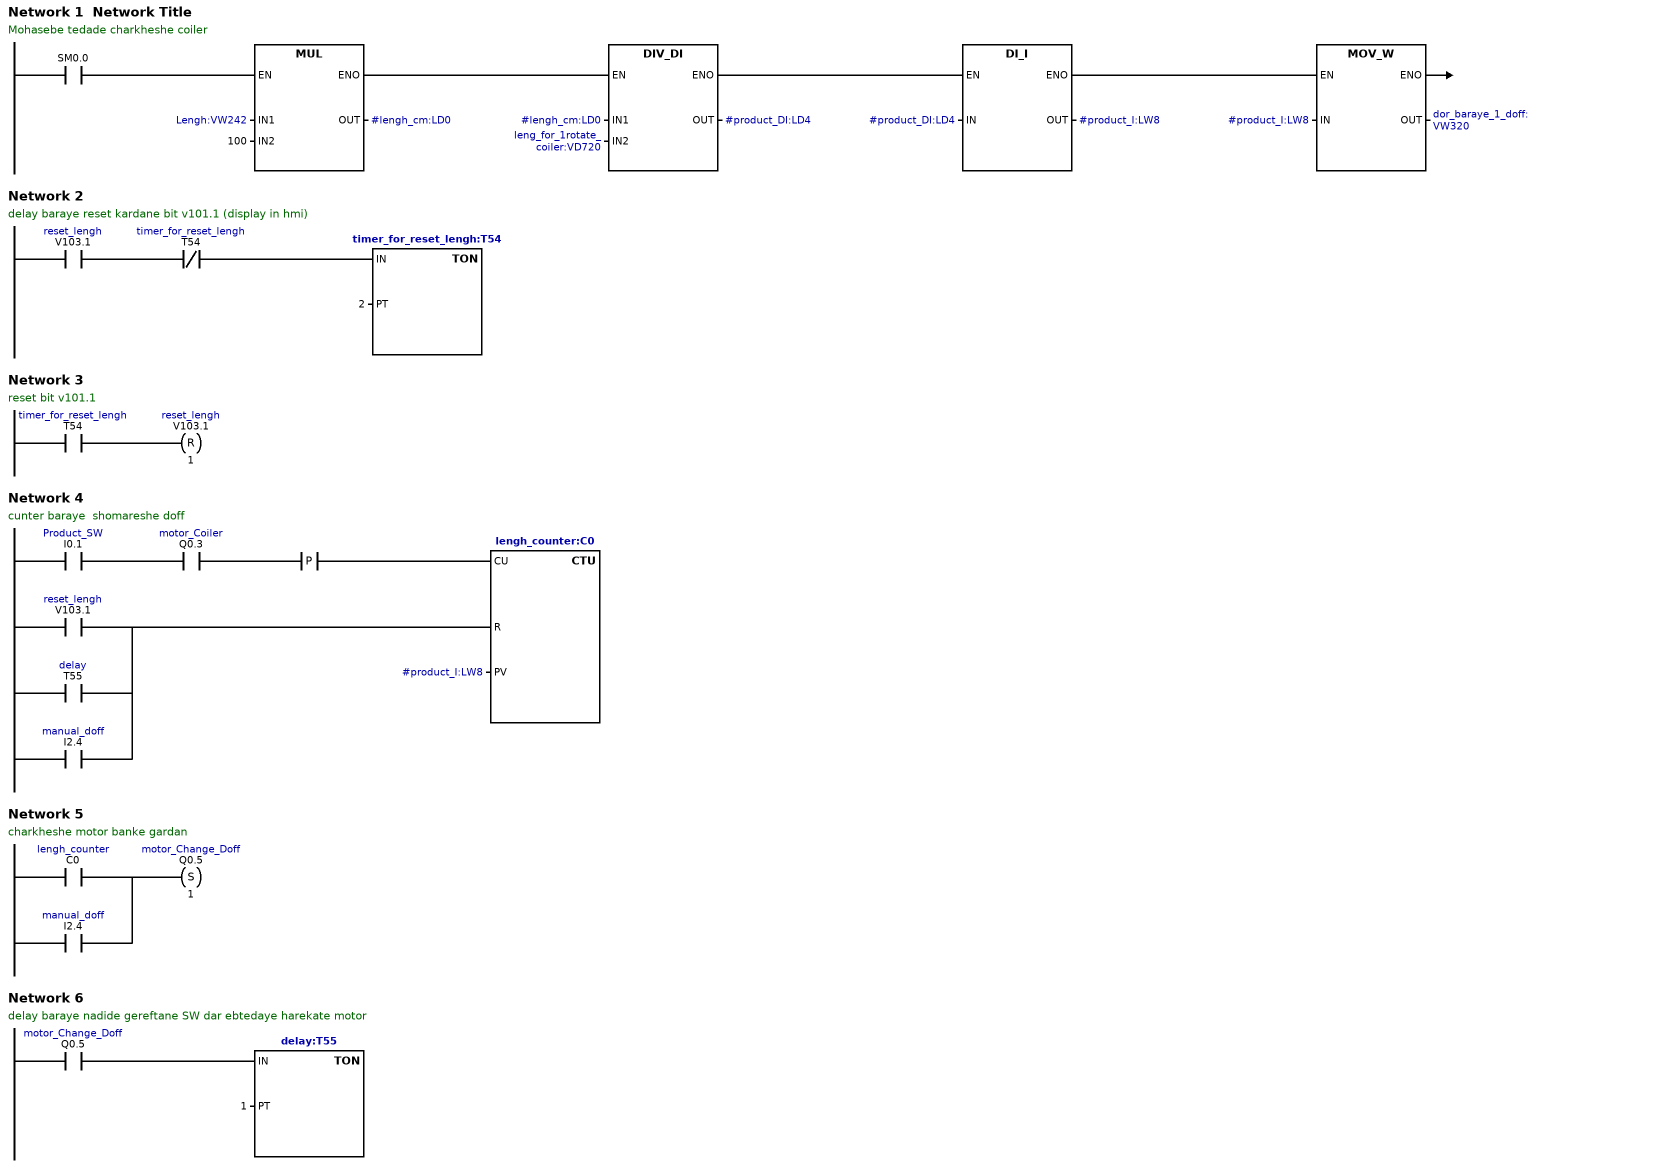
Network 1 // Network Title
// Mohasebe tedade charkheshe coiler
LD     SM0.0
MOVW   Lengh:VW242, LW2
AENO
MUL    100, #lengh_cm:LD0
AENO
MOVD   #lengh_cm:LD0, #product_DI:LD4
AENO
/D     leng_for_1rotate_coiler:VD720, #product_DI:LD4
AENO
DTI    #product_DI:LD4, #product_I:LW8
AENO
MOVW   #product_I:LW8, dor_baraye_1_doff:VW320
Network 2
// delay baraye reset kardane bit v101.1 (display in hmi)
LD     reset_lengh:V103.1
AN     timer_for_reset_lengh:T54
TON    timer_for_reset_lengh:T54, 2
Network 3
// reset bit v101.1
LD     timer_for_reset_lengh:T54
R      reset_lengh:V103.1, 1
Network 4
// cunter baraye  shomareshe doff
LD     Product_SW:I0.1
A      motor_Coiler:Q0.3
EU
LD     reset_lengh:V103.1
O      delay:T55
O      manual_doff:I2.4
CTU    lengh_counter:C0, #product_I:LW8
Network 5
// charkheshe motor banke gardan
LD     lengh_counter:C0
O      manual_doff:I2.4
S      motor_Change_Doff:Q0.5, 1
Network 6
// delay baraye nadide gereftane SW dar ebtedaye harekate motor
LD     motor_Change_Doff:Q0.5
TON    delay:T55, 1
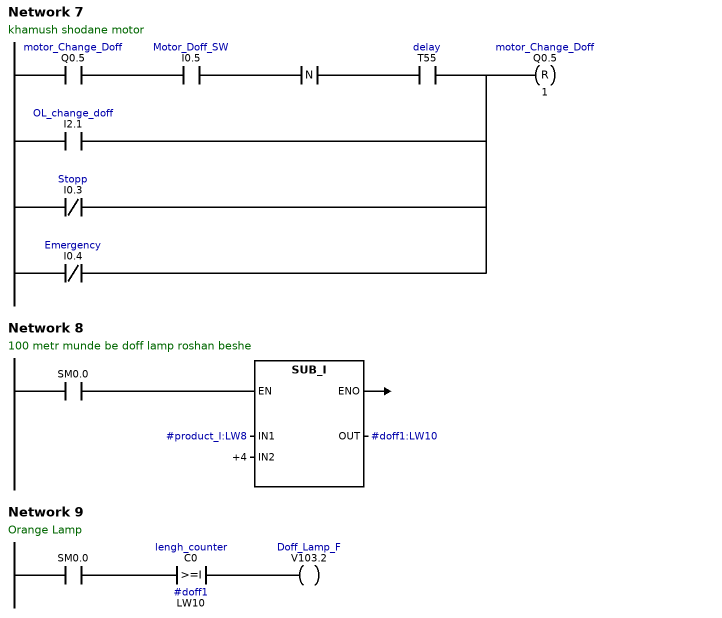
Network 7
// khamush shodane motor
LD     motor_Change_Doff:Q0.5
A      Motor_Doff_SW:I0.5
ED
A      delay:T55
O      OL_change_doff:I2.1
ON     Stopp:I0.3
ON     Emergency:I0.4
R      motor_Change_Doff:Q0.5, 1
Network 8
// 100 metr munde be doff lamp roshan beshe
LD     SM0.0
MOVW   #product_I:LW8, #doff1:LW10
-I     +4, #doff1:LW10
Network 9
// Orange Lamp
LD     SM0.0
AW>=   lengh_counter:C0, #doff1:LW10
=      Doff_Lamp_F:V103.2
END_SUBROUTINE_BLOCK

SUBROUTINE_BLOCK Amar:SBR10
TITLE=SUBROUTINE COMMENTS
VAR
hour1:INT;	// LW0 
hour:INT;	// LW2 
minute_1:INT;	// LW4 
minute:INT;	// LW6 
second_1:INT;	// LW8 
second:INT;	// LW10 
vazn_c_1:INT;	// LW12 
vazn_c_2:DINT;	// LD14 
vazn_c_3:DINT;	// LD18 
END_VAR
BEGIN
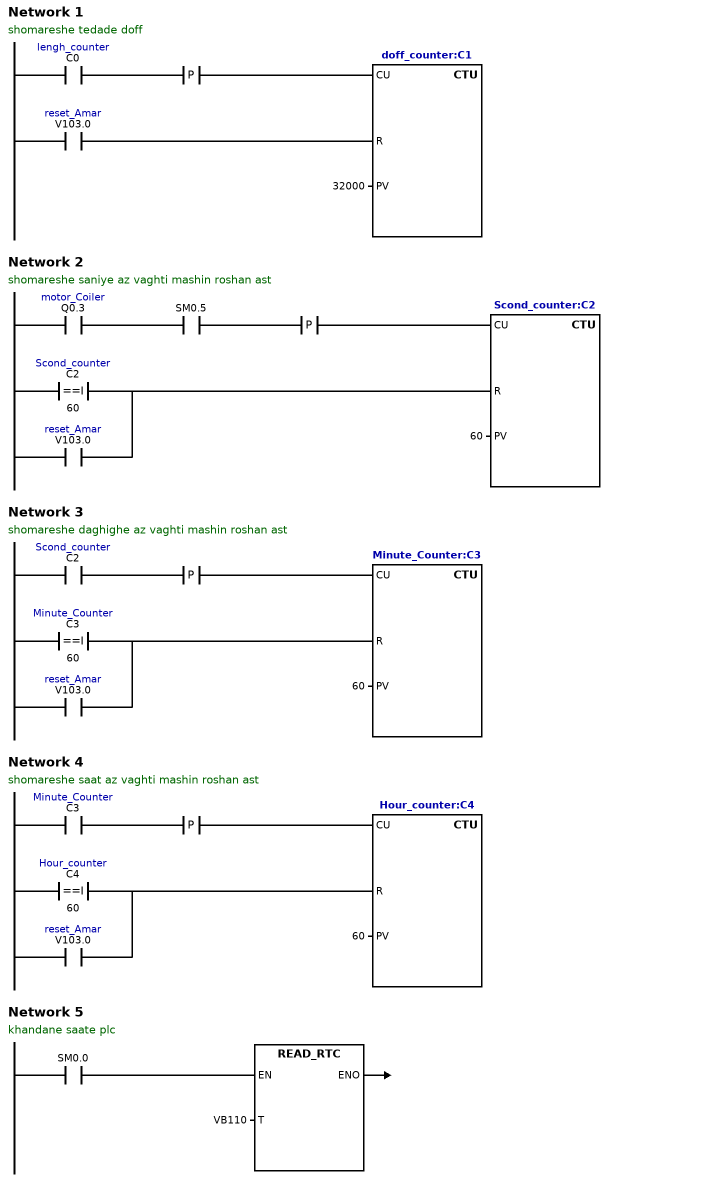
Network 1
// shomareshe tedade doff
LD     lengh_counter:C0
EU
LD     reset_Amar:V103.0
CTU    doff_counter:C1, 32000
Network 2
// shomareshe saniye az vaghti mashin roshan ast
LD     motor_Coiler:Q0.3
A      SM0.5
EU
LDW=   Scond_counter:C2, 60
O      reset_Amar:V103.0
CTU    Scond_counter:C2, 60
Network 3
// shomareshe daghighe az vaghti mashin roshan ast
LD     Scond_counter:C2
EU
LDW=   Minute_Counter:C3, 60
O      reset_Amar:V103.0
CTU    Minute_Counter:C3, 60
Network 4
// shomareshe saat az vaghti mashin roshan ast
LD     Minute_Counter:C3
EU
LDW=   Hour_counter:C4, 60
O      reset_Amar:V103.0
CTU    Hour_counter:C4, 60
Network 5
// khandane saate plc
LD     SM0.0
TODR   VB110
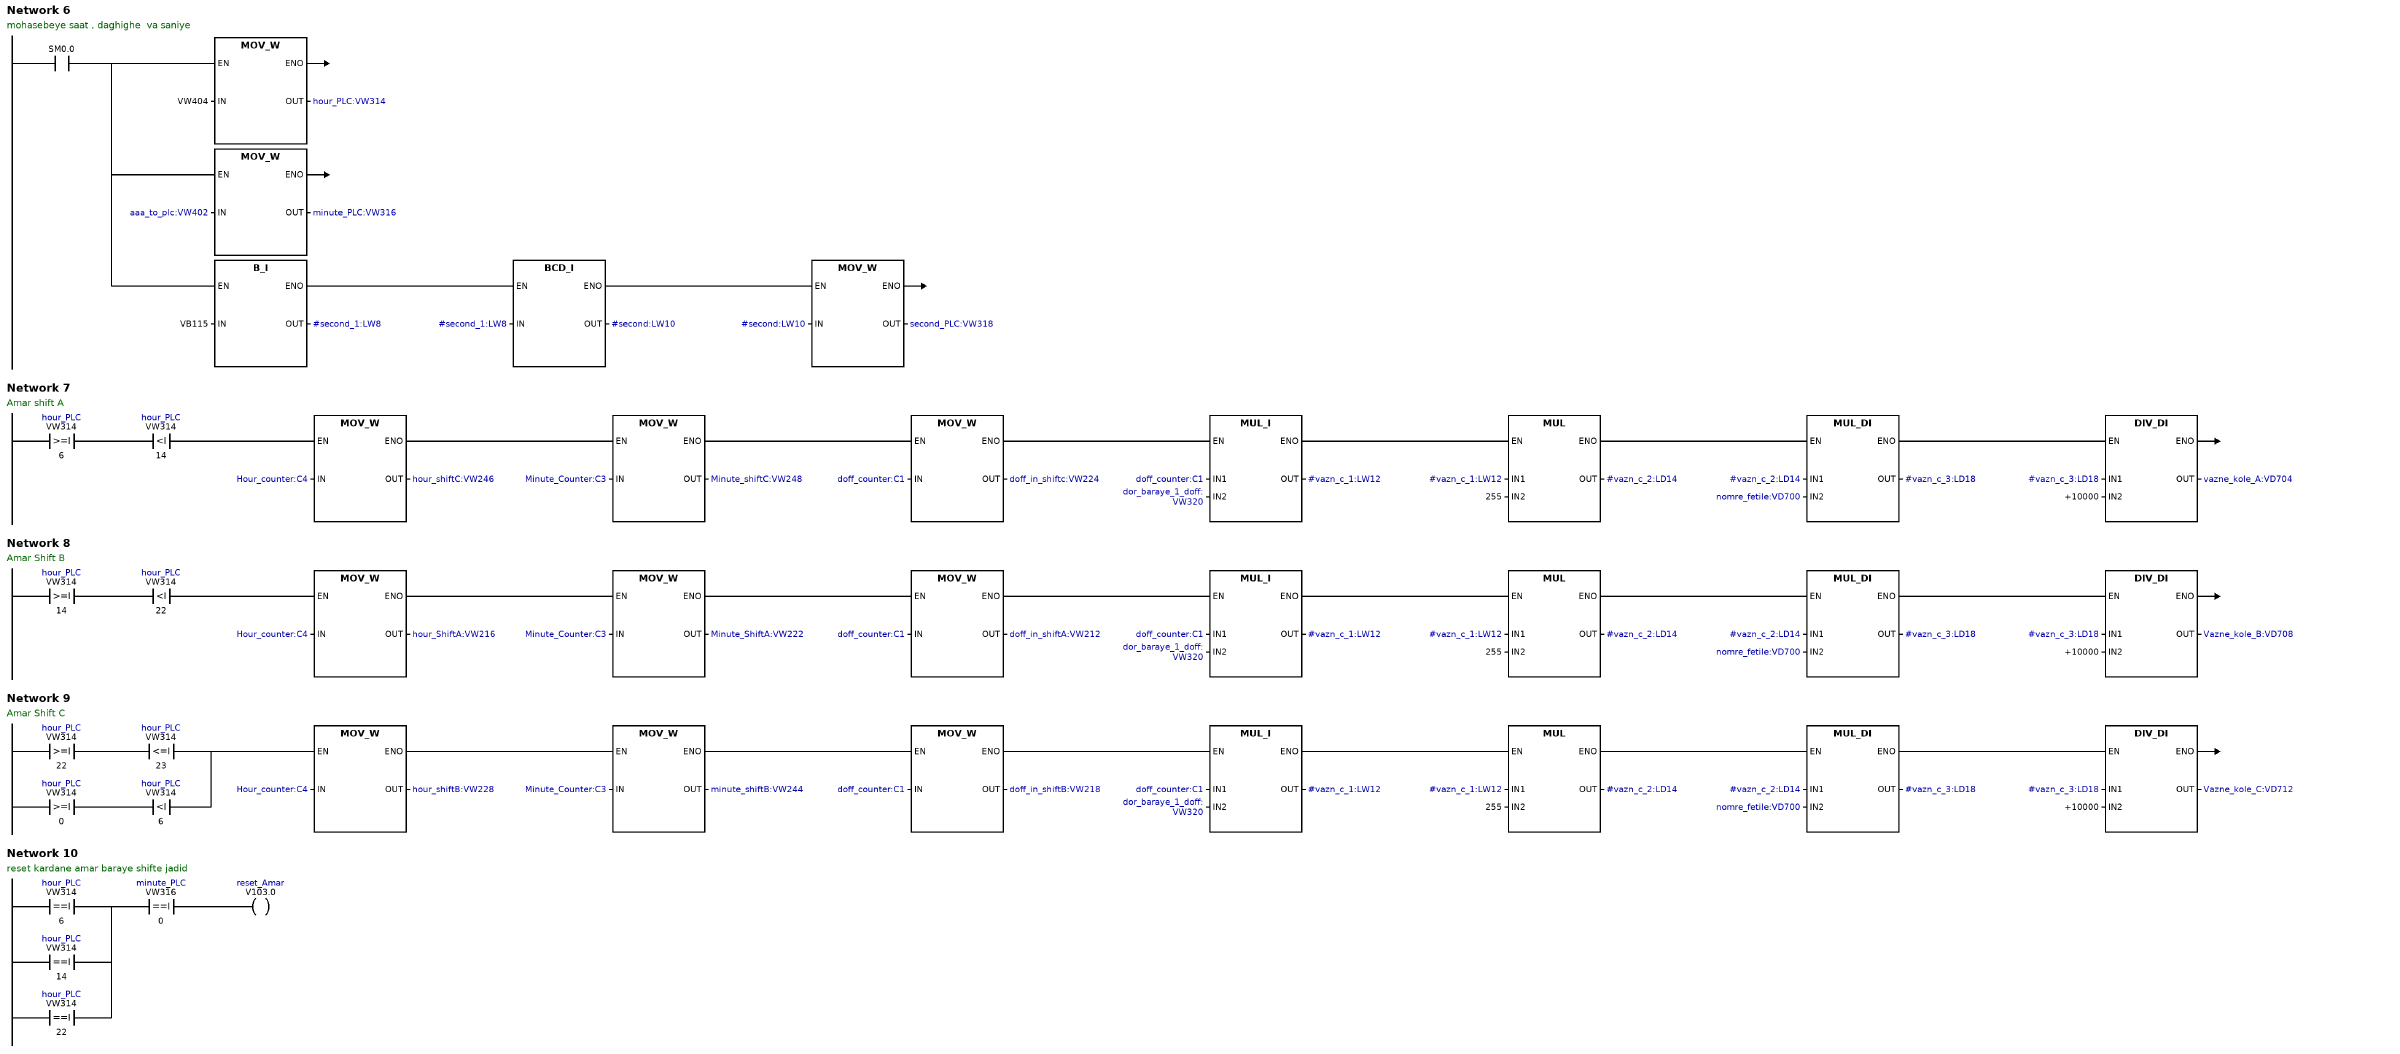
Network 6
// mohasebeye saat , daghighe  va saniye
LD     SM0.0
MOVW   VW404, hour_PLC:VW314
MOVW   aaa_to_plc:VW402, minute_PLC:VW316
BTI    VB115, #second_1:LW8
AENO
MOVW   #second_1:LW8, #second:LW10
AENO
BCDI   #second:LW10
AENO
MOVW   #second:LW10, second_PLC:VW318
Network 7
// Amar shift A
LDW>=  hour_PLC:VW314, 6
AW<    hour_PLC:VW314, 14
MOVW   Hour_counter:C4, hour_shiftC:VW246
AENO
MOVW   Minute_Counter:C3, Minute_shiftC:VW248
AENO
MOVW   doff_counter:C1, doff_in_shiftc:VW224
AENO
MOVW   doff_counter:C1, #vazn_c_1:LW12
AENO
*I     dor_baraye_1_doff:VW320, #vazn_c_1:LW12
AENO
MOVW   #vazn_c_1:LW12, LW16
AENO
MUL    255, #vazn_c_2:LD14
AENO
MOVD   #vazn_c_2:LD14, #vazn_c_3:LD18
AENO
*D     nomre_fetile:VD700, #vazn_c_3:LD18
AENO
MOVD   #vazn_c_3:LD18, vazne_kole_A:VD704
/D     +10000, vazne_kole_A:VD704
Network 8
// Amar Shift B
LDW>=  hour_PLC:VW314, 14
AW<    hour_PLC:VW314, 22
MOVW   Hour_counter:C4, hour_ShiftA:VW216
AENO
MOVW   Minute_Counter:C3, Minute_ShiftA:VW222
AENO
MOVW   doff_counter:C1, doff_in_shiftA:VW212
AENO
MOVW   doff_counter:C1, #vazn_c_1:LW12
AENO
*I     dor_baraye_1_doff:VW320, #vazn_c_1:LW12
AENO
MOVW   #vazn_c_1:LW12, LW16
AENO
MUL    255, #vazn_c_2:LD14
AENO
MOVD   #vazn_c_2:LD14, #vazn_c_3:LD18
AENO
*D     nomre_fetile:VD700, #vazn_c_3:LD18
AENO
MOVD   #vazn_c_3:LD18, Vazne_kole_B:VD708
/D     +10000, Vazne_kole_B:VD708
Network 9
// Amar Shift C
LDW>=  hour_PLC:VW314, 22
AW<=   hour_PLC:VW314, 23
LDW>=  hour_PLC:VW314, 0
AW<    hour_PLC:VW314, 6
OLD
MOVW   Hour_counter:C4, hour_shiftB:VW228
AENO
MOVW   Minute_Counter:C3, minute_shiftB:VW244
AENO
MOVW   doff_counter:C1, doff_in_shiftB:VW218
AENO
MOVW   doff_counter:C1, #vazn_c_1:LW12
AENO
*I     dor_baraye_1_doff:VW320, #vazn_c_1:LW12
AENO
MOVW   #vazn_c_1:LW12, LW16
AENO
MUL    255, #vazn_c_2:LD14
AENO
MOVD   #vazn_c_2:LD14, #vazn_c_3:LD18
AENO
*D     nomre_fetile:VD700, #vazn_c_3:LD18
AENO
MOVD   #vazn_c_3:LD18, Vazne_kole_C:VD712
/D     +10000, Vazne_kole_C:VD712
Network 10
// reset kardane amar baraye shifte jadid
LDW=   hour_PLC:VW314, 6
OW=    hour_PLC:VW314, 14
OW=    hour_PLC:VW314, 22
AW=    minute_PLC:VW316, 0
=      reset_Amar:V103.0
END_SUBROUTINE_BLOCK

SUBROUTINE_BLOCK Pulse_700ms:SBR11
TITLE=SUBROUTINE COMMENTS
BEGIN
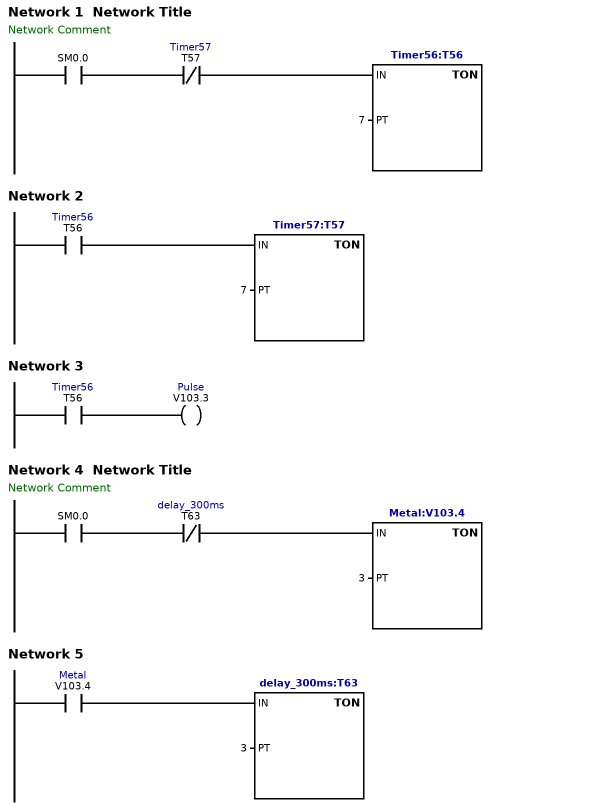
Network 1 // Network Title
// Network Comment
LD     SM0.0
AN     Timer57:T57
TON    Timer56:T56, 7
Network 2
LD     Timer56:T56
TON    Timer57:T57, 7
Network 3
LD     Timer56:T56
=      Pulse:V103.3
Network 4 // Network Title
// Network Comment
// (network saved uncompiled; LAD cells follow)
// row 0: c0 -| |- SM0.0  c1 -|/|- delay_300ms:T63  c2 --  c3 [TON Metal:V103.4 IN:=power@row0, PT:=3]
// row 1: c3 [box]
Network 5
// (network saved uncompiled; LAD cells follow)
// row 0: c0 -| |- Metal:V103.4  c1 --  c2 [TON delay_300ms:T63 IN:=power@row0, PT:=3]
// row 1: c2 [box]
END_SUBROUTINE_BLOCK
